Omron Sysmac Studio project Analogicas_Scale_HMI (Sysmac Studio 1.40.0.6, StandardProject)

# Controller new_Controller_0: NX1P2-1040DT1 version 1.13
Task PrimaryTask (priority 4, period or condition 2000): Programa0

VAR_GLOBAL
    AI0 : INT;  (* at BuiltInIO://opt/#0/Ch1_Analog_Input_Value *)
    Marcha : BOOL;
    AI0_Scale : REAL;
    Alarma : BOOL;
    AlarmaMax : BOOL;
    AlarmaMin : BOOL;
END_VAR

PROGRAM Programa0
VAR
    AI0_Limit : INT;
    AI0_Real : REAL;
    LimitAlarm1 : LimitAlarm_REAL;
    Error : BOOL;
END_VAR
VAR_EXTERNAL
    AI0 : INT;
    Marcha : BOOL;
    AI0_Scale : REAL;
    Alarma : BOOL;
    AlarmaMax : BOOL;
    AlarmaMin : BOOL;
END_VAR

(* Section Sección0: ladder, written here as Structured Text *)

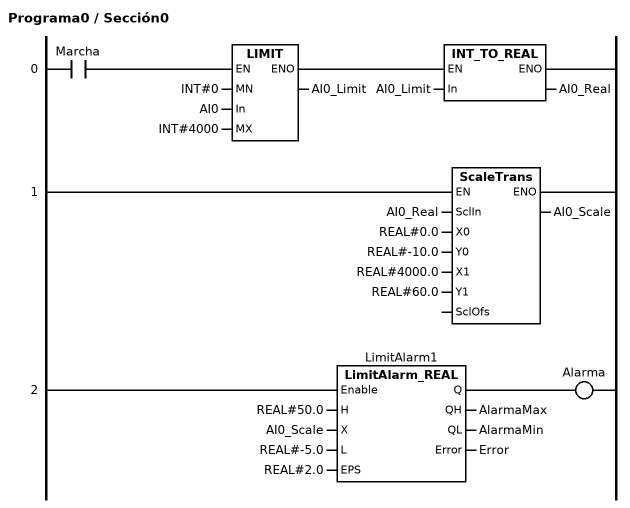
(* Rung 0 *)
IF Marcha THEN
    AI0_Limit := LIMIT(MN := INT#0, In := AI0, MX := INT#4000);
    AI0_Real := INT_TO_REAL(In := AI0_Limit);
END_IF;
(* Rung 1 *)
AI0_Scale := ScaleTrans(SclIn := AI0_Real, X0 := REAL#0.0, Y0 := REAL#-10.0, X1 := REAL#4000.0, Y1 := REAL#60.0);
(* Rung 2 *)
LimitAlarm1(Enable := TRUE, H := REAL#50.0, X := AI0_Scale, L := REAL#-5.0, EPS := REAL#2.0, QH => AlarmaMax, QL => AlarmaMin, Error => Error);
Alarma := LimitAlarm1.Q;
END_PROGRAM

# Device HMI_NA5_0 (NA): not converted